(*********************************** G.D S.p.A. - Technical Department ***********************************
============= PROGRAM INFO ============
FOLDER:             TBD
MACHINES INVOLVED:  TBD 

============= DESCRIPTION =============
csp machine declaration

============= REVISIONS ===============
Date		Version	 	Author      	Description             
----------	-------		------------  	--------------------------------------------
2019/04/05 	0000.00	 	M.Grasso		Creation of the PRG
2020/05/04 	0000.01	 	G.Imbriaco		From original author, G.Imbriaco: AccU Change motor with absolute encoder and brake.
										If position_req_mm parameter different from actual_pos_mm and machine reset_edge
										the motor move to position_req then disable again
										Manual movement with basc axis object under test( preset, moving,...)
										All disabled if main accU_Change is not Operational

**********************************************************************************************************)
(*$R process_ref := prc; $*)
PROGRAM csp_transfer_accumulator_accU_convDepth
VAR
	
	prc:											process;
	prc_path:										STRING;
	
	axis:											axis;
	Slot89_drv:										coe_drive;

	not_in_position:								message;
	axis_restore_absolute_position_fb:				restore_absolute_position_with_retain_fb;


	disable_req:									BOOL:=FALSE;
	position_req:									LREAL:=0.0;(*$P $*)
	move_velocity_req:								LREAL:=10.0;(*$P $*)
	position_req_tolerance:							LREAL:=0.2;	(*$P $*)
	
	axis_status:									axis_status_enum := AXIS_STATUS_PARAMETERS_START;(*$M $*)
	in_position:									BOOL:=FALSE;(*$M $*)	
	actual_position:								LREAL:=0.0; (*$M $*)
	axis_move_condition:							BOOL:=FALSE;
	torque_limit:                                   INT := 5000;    
    torque_limit_old:                               INT;
	
	in_position_motcond:							motorization_conditioner;
	fsm_status:										csp_transfer_accumulator_accU_convDepth_enum;(*$M $*)
	fsm_next_status:								csp_transfer_accumulator_accU_convDepth_enum;
	fsm_enable_condition:							BOOL:=FALSE;
	debug_state_machine:							BOOL:=FALSE;
	debug_state_machine_one_step:					BOOL:=FALSE;
	NC_encoder_val AT %I*:							DINT;
	
	temp_accel:										LREAL:= 100;
	temp_decel:										LREAL:= 100;
	temp_jerk:										LREAL:= 10000;
	
END_VAR
VAR PERSISTENT
	axis_restore_absolute_position_data:			restore_absolute_position_with_retain_struct;
END_VAR

_read_var_input();

_object_manager();

IF NOT objects_running()
THEN
	RETURN;	
END_IF

_read_process_image();

_mode_manager();

CASE process_get_mode(prc) OF
	MODE_ABSENT,
	MODE_INACTIVE:
		RETURN;
	MODE_TEST:
		_handle_process_test();
END_CASE

_set_runtime_properties();

(********************************* BODY *********************************)
//Axis Torque Limit
IF torque_limit <> Torque_limit_old
THEN
    IF coe_drive_write_parameter(
        index:=16#7010 ,
        complete_access:= FALSE ,
        sub_index:= 16#0B,
        data_source:= ADR(torque_limit),
        data_lenght:= SIZEOF(torque_limit),
        CONVERSION_this:=csp_transfer_accumulator_accU_convDepth.axis.coe_drive^ ) = COE_DRIVE_RETURN_VALUE_DONE
        THEN
		torque_limit_old := Torque_limit;
	END_IF
END_IF 

//Axis move condition
IF 	csp_main_accuChange.transfer_accumulator_accU_depth_move_req 
	OR jog_manager_is_jog_axis_active(SMTR61720_SMTR61730_TRANSFER_ACCUMULATOR_DEPTH_AND_CONVEYOR_DEPTH, csp_main_jogManager.jog_manager_accuchange)
THEN
	axis_move_condition := TRUE;
ELSE
	axis_move_condition := FALSE;
END_IF

(*FSM Control*)
fsm_enable_condition := axis_is_ok(FALSE, axis)
						(*AND
						process_is_ready(prc) *)
						AND
						process_subtree_is_ready(prc)
						AND
						process_get_mode(csp_main_accuChange.prc) = MODE_OPERATIONAL					
						AND
						axis_restore_absolute_position_fb.o_position_restored					
						AND
						NOT disable_req;		
					
IF	(NOT fsm_enable_condition
	OR
	disable_req)
	AND
	fsm_status <> CSP_TRANSFER_ACCUMULATOR_ACCU_CONV_DEPTH_STATUS_DISABLED
	AND
	fsm_status < CSP_TRANSFER_ACCUMULATOR_ACCU_CONV_DEPTH_STATUS_STOP_REQUEST
THEN
	fsm_status	:=	CSP_TRANSFER_ACCUMULATOR_ACCU_CONV_DEPTH_STATUS_STOP_REQUEST;
END_IF


CASE fsm_status OF
	
	CSP_TRANSFER_ACCUMULATOR_ACCU_CONV_DEPTH_STATUS_NOT_INITIALIZED:
	
        IF	axis_is_ok(return_when_absent := TRUE, CONVERSION_this := axis)
        THEN
            fsm_next_status := CSP_TRANSFER_ACCUMULATOR_ACCU_CONV_DEPTH_STATUS_DISABLED;
        END_IF

		
	CSP_TRANSFER_ACCUMULATOR_ACCU_CONV_DEPTH_STATUS_DISABLED:
	
		IF	fsm_enable_condition
		THEN
			(* Axis with absolute encoder, no home procedure request *)
			fsm_next_status := CSP_TRANSFER_ACCUMULATOR_ACCU_CONV_DEPTH_STATUS_POSITION_CHECK;
		END_IF;
	
		
	CSP_TRANSFER_ACCUMULATOR_ACCU_CONV_DEPTH_STATUS_POSITION_CHECK:

		IF 	axis_move_condition
			OR jog_manager_is_jog_axis_active(SMTR61720_SMTR61730_TRANSFER_ACCUMULATOR_DEPTH_AND_CONVEYOR_DEPTH, csp_main_jogManager.jog_manager_accuchange)
		THEN
			fsm_next_status := CSP_TRANSFER_ACCUMULATOR_ACCU_CONV_DEPTH_STATUS_ENABLE_REQUEST;
		END_IF			
	
		
	CSP_TRANSFER_ACCUMULATOR_ACCU_CONV_DEPTH_STATUS_ENABLE_REQUEST:
	
		axis_enable(axis);
		IF axis_is_standstill(axis)
		THEN
			fsm_next_status	:=	CSP_TRANSFER_ACCUMULATOR_ACCU_CONV_DEPTH_STATUS_ENABLED;
		END_IF		

		
	CSP_TRANSFER_ACCUMULATOR_ACCU_CONV_DEPTH_STATUS_ENABLED:
	
		IF 	axis_move_condition 
			OR jog_manager_is_jog_axis_active(SMTR61720_SMTR61730_TRANSFER_ACCUMULATOR_DEPTH_AND_CONVEYOR_DEPTH, csp_main_jogManager.jog_manager_accuchange)
		THEN
			fsm_next_status	:= CSP_TRANSFER_ACCUMULATOR_ACCU_CONV_DEPTH_STATUS_GEAR_REQUEST;	
		END_IF
			
		
	CSP_TRANSFER_ACCUMULATOR_ACCU_CONV_DEPTH_STATUS_GEAR_REQUEST:

		IF	axis_is_standstill(axis)
			AND (csp_transfer_accumulator_accU_virtualMaster.master_redefined
			OR jog_manager_is_jog_axis_active(SMTR61720_SMTR61730_TRANSFER_ACCUMULATOR_DEPTH_AND_CONVEYOR_DEPTH, csp_main_jogManager.jog_manager_accuchange))
		THEN
			axis_engage_position_gear(
				ratio 			:= 1.0,
				acceleration 	:= temp_accel,//csp_main_accuChange.CONSTANTS.MAX_ACCELERATION_MMpSEC2,
				deceleration 	:= temp_decel,//csp_main_accuChange.CONSTANTS.MAX_DECELERATION_MMpSEC2,
				jerk			:= temp_jerk,//csp_main_accuChange.CONSTANTS.MAX_JERK_MMpSEC3,
				master 			:= csp_transfer_accumulator_accU_virtualMaster.axis,
				CONVERSION_this := axis);			
		END_IF
		
		IF axis_is_gear_engaging(axis)
		THEN
			fsm_next_status	:=	CSP_TRANSFER_ACCUMULATOR_ACCU_CONV_DEPTH_STATUS_GEARING;
		END_IF

		
	CSP_TRANSFER_ACCUMULATOR_ACCU_CONV_DEPTH_STATUS_GEARING:
		
		IF axis_is_gear_engaged(axis)
		THEN
			fsm_next_status	:=	CSP_TRANSFER_ACCUMULATOR_ACCU_CONV_DEPTH_STATUS_GEARED;
		END_IF
		
		
	CSP_TRANSFER_ACCUMULATOR_ACCU_CONV_DEPTH_STATUS_GEARED:
			
		IF axis_is_moving(csp_transfer_accumulator_accU_virtualMaster.axis)
		THEN
			fsm_next_status := CSP_TRANSFER_ACCUMULATOR_ACCU_CONV_DEPTH_STATUS_MOVING;
		END_IF
		
		(* BREAKS GEAR IF NOT JOGGING *)
		IF 	NOT csp_main_accuchange.Brand_Change_Occurred
			AND NOT jog_manager_is_jog_axis_active(SMTR61720_SMTR61730_TRANSFER_ACCUMULATOR_DEPTH_AND_CONVEYOR_DEPTH, csp_main_jogManager.jog_manager_accuchange)
		THEN
			fsm_next_status := CSP_TRANSFER_ACCUMULATOR_ACCU_CONV_DEPTH_STATUS_STOP_REQUEST;
		END_IF
	
		
	CSP_TRANSFER_ACCUMULATOR_ACCU_CONV_DEPTH_STATUS_MOVING:

		IF NOT axis_move_condition
			OR ( 
			csp_transfer_accumulator_accU_virtualMaster.fsm_status <> CSP_TRANSFER_ACCUMULATOR_ACCU_VIRTUAL_MASTER_STATUS_ABS_MOVING (* Disables if master disable *)
			AND
			NOT jog_manager_is_jog_axis_active(SMTR61720_SMTR61730_TRANSFER_ACCUMULATOR_DEPTH_AND_CONVEYOR_DEPTH, csp_main_jogManager.jog_manager_accuchange)	
				)					
		THEN
			fsm_next_status := CSP_TRANSFER_ACCUMULATOR_ACCU_CONV_DEPTH_STATUS_STOP_REQUEST;
		END_IF
		
		
	CSP_TRANSFER_ACCUMULATOR_ACCU_CONV_DEPTH_STATUS_DISENGAGE_TO_RECOVER_TO_MASTER:
	
		axis_disengage(
			mode := AXIS_DISENGAGE_AND_STOP,
			position := 0,
			velocity := 2,
			acceleration := csp_main_accuChange.CONSTANTS.MAX_ACCELERATION_MMpSEC2,
			deceleration := csp_main_accuChange.CONSTANTS.MAX_DECELERATION_MMpSEC2,
			jerk := csp_main_accuChange.CONSTANTS.MAX_JERK_MMpSEC3,
			CONVERSION_this := axis);
		
		IF axis_is_disengaged(axis)
		THEN
			fsm_next_status := CSP_TRANSFER_ACCUMULATOR_ACCU_CONV_DEPTH_STATUS_RECOVER_TO_MASTER;
		END_IF
		
		
	CSP_TRANSFER_ACCUMULATOR_ACCU_CONV_DEPTH_STATUS_RECOVER_TO_MASTER:
	
		 axis_move_absolute(
			position 		:= position_req,
			velocity 		:= move_velocity_req,
			direction		:= AXIS_SHORTEST_WAY,
			acceleration 	:= csp_main_accuChange.CONSTANTS.MAX_ACCELERATION_MMpSEC2,
			deceleration 	:= csp_main_accuChange.CONSTANTS.MAX_DECELERATION_MMpSEC2,
			jerk 			:= csp_main_accuChange.CONSTANTS.MAX_JERK_MMpSEC3, 
			buffer_mode 	:= AXIS_BUFFER_MODE_ABORTING,
			CONVERSION_this := axis
			); 
			
		IF NOT axis_move_condition
		THEN
			fsm_next_status := CSP_TRANSFER_ACCUMULATOR_ACCU_CONV_DEPTH_STATUS_STOP_REQUEST;
		END_IF
		
		
	CSP_TRANSFER_ACCUMULATOR_ACCU_CONV_DEPTH_STATUS_STOP_REQUEST:

		axis_stop(
		    deceleration 	:= csp_main_accuChange.CONSTANTS.MAX_DECELERATION_MMpSEC2,
		    jerk 			:= csp_main_accuChange.CONSTANTS.MAX_JERK_MMpSEC3,
		    CONVERSION_this 			:= axis);

		IF 	axis_is_standstill(axis)
			OR
			NOT axis_is_ok(FALSE, axis)
			OR
			axis_is_disabled(axis)
		THEN
			fsm_next_status := CSP_TRANSFER_ACCUMULATOR_ACCU_CONV_DEPTH_STATUS_DISABLE_REQUEST;
		END_IF
		

	CSP_TRANSFER_ACCUMULATOR_ACCU_CONV_DEPTH_STATUS_DISABLE_REQUEST:
	
   		axis_disable(axis);
        IF	axis_is_disabled(axis)
        THEN
            fsm_next_status := CSP_TRANSFER_ACCUMULATOR_ACCU_CONV_DEPTH_STATUS_DISABLED;
        END_IF;

END_CASE;

IF NOT debug_state_machine
	OR
	debug_state_machine_one_step
THEN
	fsm_status := fsm_next_status;
	debug_state_machine_one_step := FALSE;
END_IF

(************************************************************************)
_brand_change();

_handle_messages();

_write_output();

ACTION _brand_change:

END_ACTION

ACTION _handle_messages:
IF in_position OR csp_main_jogManager.jog_is_active
THEN
	;//process_message_reset(not_in_position);
ELSE
	IF csp_main_accuChange.machine_size_complete = FALSE
	THEN
		;//process_message_reset(not_in_position);
	ELSE
		;//process_message_set(errorID_1:= 1, errorID_2:= 0, errorID_3:= 0, CONVERSION_this:= not_in_position);
	END_IF
END_IF
END_ACTION

ACTION _handle_process_test:
;
END_ACTION

ACTION _mode_manager:
IF process_mode_req_is_pending(prc)
THEN
    process_apply_mode_req_first_step(prc);
    CASE process_get_mode(prc) OF
        MODE_TO_ABSENT:
			;
        MODE_TO_INACTIVE:
			;
        MODE_TO_TEST:
			;
        MODE_TO_OPERATIONAL:
			;
    END_CASE
    process_apply_mode_req_second_step(prc);
END_IF
END_ACTION

ACTION _object_manager:
IF objects_initialization()
THEN
	sub_process_init(
		object_name								:= 'csp_transfer_accumulator_accU_convDepth.prc', 
		process									:= csp_transfer_accumulator_accU.prc, 
		CONVERSION_this							:= prc);
		
	prc_path 									:= process_get_path(prc);
	
	IF csp_main_configurator.Physical_hw 
	THEN
		axis_init(
			object_name							:= CONCAT(prc_path, '_axis'), 
			axis_type							:= AXIS_TYPE_SERVO, 
			encoder_scaling_factor				:= 0.15*0.00000095367431640625,
			modulo								:= 1024, 
  			process								:= prc, 
			CONVERSION_this						:= axis);
						
		axis_init_absolute_encoder_preset(   
        	position                    		:=    200,
        	CONVERSION_this                		:=    axis);

		axis_add_safety_integrated_series(
			safety_integrated_series			:= csp_transfer_main_safety_accUChange.sis,
			CONVERSION_this						:= axis);
		axis_set_brake_type(AXIS_BRAKE_DRIVE_CMD, axis);
	ELSE
		axis_init(
			object_name 						:= CONCAT(prc_path, '_axis'),
			axis_type 							:= AXIS_TYPE_VIRTUAL,
			encoder_scaling_factor 				:= G_VIRTUAL_ENCODER_SCALING_FACTOR_DEGPINC,
			modulo 								:= 0,
			process 							:= prc,
			CONVERSION_this 					:= axis);
	END_IF
	
	axis_set_rotation_direction(
		invert_encoder_counting					:= FALSE,
		invert_motor_polarity					:= FALSE,
		CONVERSION_this							:= axis);

	coe_drive_init(
		object_name 							:= CONCAT(prc_path, '_Slot89_drv'),
		device_name 							:= 'IO61600Slot89 (EL7211)',
		vendor 									:= DRIVE_BECKHOFF_EL72x1,
		mode 									:= COE_DRIVE_MODE_DRIVEN_BY_AXIS,
		ethercat_master							:= csp_main.cabinet_transfer_ethercat_master,
		process									:= prc,
		CONVERSION_this 						:= Slot89_drv);

	axis_add_coe_drive(
		coe_drive								:= Slot89_drv,
		CONVERSION_this							:= axis);
		
	axis_set_max_dynamic(
		reference_velocity						:=	csp_main_accuChange.CONSTANTS.MAX_VELOCITY_MMpSEC,
		velocity								:=	csp_main_accuChange.CONSTANTS.MAX_VELOCITY_MMpSEC,
		acceleration							:=	csp_main_accuChange.CONSTANTS.MAX_ACCELERATION_MMpSEC2,
		deceleration							:=	csp_main_accuChange.CONSTANTS.MAX_DECELERATION_MMpSEC2,
		jerk									:=	csp_main_accuChange.CONSTANTS.MAX_JERK_MMpSEC3,
		following_error							:=	csp_main_accuChange.CONSTANTS.MAX_FOLLOWING_ERROR_MM,
		CONVERSION_this							:=	axis);

	process_message_init(
		object_name:= CONCAT(prc_path, '_not_in_position'), 
		behaviour:= MESSAGE_BEHAVIOUR_STATE, 
		reset_timeout:= 0, 
		disableable:= TRUE, 
		individual_reset:= FALSE, 
		machine_reaction:= MACHINE_REACTION_STOP_IN_PHASE_ONE, 
		typology:= MESSAGE_TYPOLOGY_ABNORMAL, 
		process:= prc, 
		CONVERSION_this:= not_in_position);
END_IF

IF objects_running()
THEN
	process_cycle(prc);
	axis_cycle(axis);
	coe_drive_cycle(Slot89_drv);
END_IF
END_ACTION

ACTION _read_process_image:
axis_restore_absolute_position_fb(
	io_retain_data				:= axis_restore_absolute_position_data, 
	io_axis						:= axis);
END_ACTION

ACTION _read_var_input:
;
END_ACTION

ACTION _set_runtime_properties:

axis_status := axis_get_status(axis);
actual_position :=axis_get_actual_incremental_position(axis); (* axis_get_actual_modulo_position(axis); only with modulo*)

IF (ABS(csp_transfer_accumulator_accu_depth.position_req - actual_position) < position_req_tolerance) //+ csp_transfer_accumulator_accu_virtualMaster.dif_depth_and_convDepth) < position_req_tolerance
	OR process_get_mode(prc)= MODE_ABSENT
	OR process_get_mode(csp_main_accuChange.prc) = MODE_ABSENT
THEN
	in_position := TRUE;
ELSE
	in_position := FALSE;	
END_IF
END_ACTION

ACTION _write_output:
;
END_ACTION

END_PROGRAM

(* stored: Version 1.1.0.1, ProductVersion 3.1.4024.3
   POU csp_transfer_accumulator_accU_convDepth: Id {40249a03-7279-483f-aae0-1bed69097a95}, SpecialFunc None
   Action _brand_change: Id {936bdcb7-ae00-4431-adef-75b680e9edb2}
   Action _handle_messages: Id {4e9e13bb-faed-44af-9b97-cbe99302daf0}
   Action _handle_process_test: Id {4fa85aec-805f-4698-abdc-079f2276d44c}
   Action _mode_manager: Id {17a55c79-b2a5-4478-9400-cb0caf82793d}
   Action _object_manager: Id {4c55c567-cfb8-43b7-939b-c87f3a5336cf}
   Action _read_process_image: Id {0b4a1ee1-acb8-4ca1-b364-b7490f160cdd}
   Action _read_var_input: Id {1daaed66-1785-4dee-8ea9-719bfbd78df2}
   Action _set_runtime_properties: Id {6db8e376-5f26-467a-9c0b-f3ed00195c8e}
   Action _write_output: Id {ca47b10e-064b-4a3e-a51e-b66e6855505a} *)
